TYPE ST_ReturnStructure :
STRUCT
	Done	: BOOL;
	Active	: BOOL;
	Busy	: BOOL;
	Aborted	: BOOL;
	Error	: BOOL;
	ErrorId	: UDINT;
END_STRUCT
END_TYPE

(* stored: Version 1.1.0.1, ProductVersion 3.1.4026.19
   DUT ST_ReturnStructure: Id {3a2f6e92-255e-4004-a2a9-b66ff22b6eb8} *)
